// TIA Portal V20 export
// export: Created 2025-12-01T14:57:04.3454128Z, ExportSetting None, DisplayName Totally Integrated Automation Portal, DisplayVersion V20 Update 3, DisplayName TIA Portal Openness, DisplayVersion V20 Update 3, DisplayName TIA Portal Version Control Interface, DisplayVersion V20 Update 3, DisplayName STEP 7 Professional, DisplayVersion V20 Update 3, DisplayName STEP 7 Safety, DisplayVersion V20 Update 2, DisplayName WinCC Basic/Comfort/Advanced, DisplayVersion V20 Update 3, DisplayName WinCC Professional, DisplayVersion V20 Update 3, DisplayName WinCC Unified, DisplayVersion V20 Update 3
FUNCTION "FC778_TipoCajaPlastico_EnMesaApilador" : Void   // FC778, STL
TITLE = Informacion del tipo de Caja en la Mesa
{ S7_Optimized_Access := 'FALSE' }
AUTHOR : TRACKING
NAME : 01032013
VERSION : 3.0
// stored: AutoNumber false
   VAR_INPUT
      Mesa : UInt;   // Numero de Mesa
   END_VAR
   VAR_OUTPUT
      DosCajas : Bool;   // Hay dos Cajas en la Mesa
      CajaPequena : Bool;   // Caja Primera Pequeña
      CajaGrande : Bool;   // Caja Segunda Pequeña
   END_VAR
   VAR_TEMP
      NumeroUT : UInt;
      SiguienteUT : UInt;
      AnteriorUT : UInt;
      GrupoUT : UInt;   // Grupo de la UT
   END_VAR
BEGIN

NETWORK
TITLE = Inicialializar
////////////////////////////////////////////////////////////////////////////
// --- Inicializar Variables

      SET;
      R     #DosCajas;
      R     #CajaPequena;
      R     #CajaGrande;



NETWORK
TITLE = Calculo de Activacion
////////////////////////////////////////////////////////////////////////////
// --- Ver si hay UT's en la Mesa


      L     "DB810_ColasMesas".Colas[#Mesa].UT_PrimeraMesa;
      T     #SiguienteUT;

      L     #SiguienteUT;  // - Si no hay UT's
      L     0;
      ==I;
      JC    Final;


////////////////////////////////////////////////////////////////////////////
// --- Buscar la Ultima UT de la Mesa

SeguirBuscandoUltimaUT:NOP   0;
      L     #SiguienteUT;
      T     #NumeroUT;

      L     "DB812_UTs_Control".UT[#NumeroUT].UT_SiguienteMesa;
      T     #SiguienteUT;

      L     #SiguienteUT;  // Es la Ultima UT de la Mesa ?
      L     0;
      <>I;
      JC    SeguirBuscandoUltimaUT;

// --- Encontrada la Ultima


////////////////////////////////////////////////////////////////////////////
// --- Mirar el Tipo de Caja - Ultima UT de la Mesa

      L     "DB812_UTs_Control".UT[#NumeroUT].Grupo;
      T     #GrupoUT;

      L     "DB812_UTs_Control".UT[#NumeroUT].TipoCarga;  // TipoCaja - Posicion 28
      L     10;
      /I;
      L     10;  // CajaPequeña (3x)
      ==I;
      JC    CajaDeTipoPequeno;
      JU    CajaDeTipoGrande;


////////////////////////////////////////////////////////////////////////////
// --- Tipo de Caja Grande
CajaDeTipoGrande:NOP   0;
      SET;
      S     #CajaGrande;
      JU    Final;


////////////////////////////////////////////////////////////////////////////
// --- Tipo de Caja Pequeño
CajaDeTipoPequeno:NOP   0;
      SET;
      S     #CajaPequena;

// --- Mirar si es una Doble Caja Pequeña en la Fila

      L     "DB812_UTs_Control".UT[#NumeroUT].UT_AnteriorMesa;
      T     #AnteriorUT;

      L     #AnteriorUT;
      L     0;
      ==I;
      JC    Final;  // Hay mas UT's en la Mesa ?

      L     "DB812_UTs_Control".UT[#AnteriorUT].Grupo;
      L     #GrupoUT;
      <>I;
      JC    Final;

      SET;
      S     #DosCajas;  // Hay dos cajas en la Mesa



NETWORK
TITLE = Final de la Funcion
////////////////////////////////////////////////////////////////////////////
// --- Final de la Funcion
Final:NOP   0;


END_FUNCTION
